PROGRAM MAIN
VAR
	vacSensor : FB_VacSensor;
END_VAR

vacSensor();

END_PROGRAM

(* stored: Version 1.1.0.1
   POU MAIN: Id {8930809c-2430-4d4a-8075-59855ac3ebfc}, SpecialFunc None *)
